KUKA KRL program: exemplo_1.src

&ACCESS RVP
&REL 1
DEF hello()
  MsgNotify("Olá Mundo")
END
